Fanuc KAREL source: compact_preamble.KL

PROGRAM KB00142
%NOLOCKGROUP
VAR
P1 : STRING[80];P2:INTEGER;P3:INTEGER;P4:INTEGER
BEGIN
P1='A'
P2=1
P3=1
P4=1
PUSH_KEY_RD(P1,P2,P3,P4)
END KB00142
